Staubli VAL3: XHS3023L.dtx

public frame fCadToReal = {fatherId=fUserFrame[0]}
public frame fUserFrame = {fatherId=world[0]}
public mdesc mNomSpeed = {blend=off}
public tool tTool = {x=968, y=-155, z=-238, rx=-90, rz=180, fatherId=flange[0], ioLink=valve1}
